(* CoDeSys 2.3.9.50 project: 4D.pr6 *)
(* Libraries: STANDARD.LB6 5.6.98 12:03:02 *)

(* POU MAIN, LD *)
PROGRAM MAIN
VAR
	Stacking AT %IX0.0: BOOL;
	C1: CTU;
	C2: CTU;
	C3: CTU;
	StackProcess AT %QX0.0: BOOL;
	Space AT %QX0.2: BOOL;
	A AT %IX0.3: BOOL;
	t1: TON;
	Banded AT %QX0.3: BOOL;
END_VAR
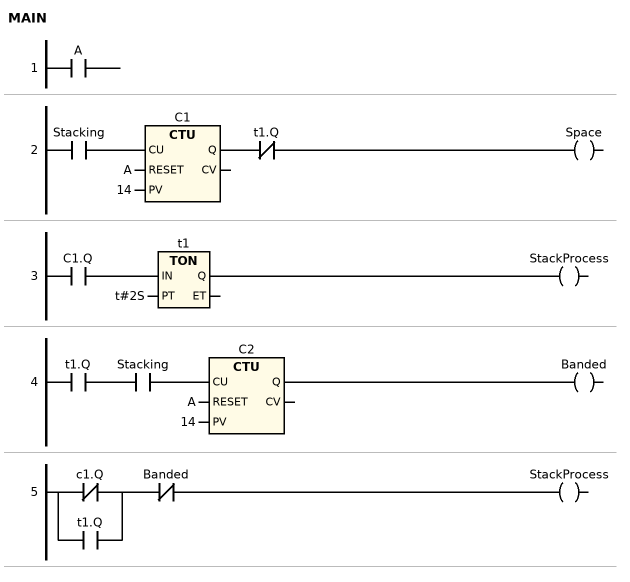
_LD_ (* Ladder Diagram *)
NETWORK 1
	[A]
NETWORK 2
	[Stacking] - C1:CTU(CU: *, RESET: A, PV: 14) - [/t1.Q] --- (Space)
NETWORK 3
	[C1.Q] - t1:TON(IN: *, PT: t#2S) --- (StackProcess)
NETWORK 4
	[t1.Q] - [Stacking] - C2:CTU(CU: *, RESET: A, PV: 14) --- (Banded)
NETWORK 5
	{ [/c1.Q] | [t1.Q] } - [/Banded] --- (StackProcess)
_END_LD_
(* the same logic as Structured Text *)
(* Network 1 *)
(* Network 2 *)
C1(CU := Stacking, RESET := A, PV := 14);
Space := C1.Q AND NOT t1.Q;
(* Network 3 *)
t1(IN := C1.Q, PT := t#2S);
StackProcess := t1.Q;
(* Network 4 *)
C2(CU := t1.Q AND Stacking, RESET := A, PV := 14);
Banded := C2.Q;
(* Network 5 *)
StackProcess := (NOT c1.Q OR t1.Q) AND NOT Banded;
END_PROGRAM
